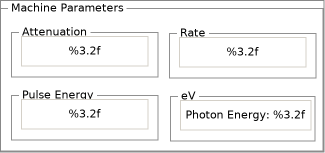
VISUALIZATION BeamParameterStats  // 325x153
VAR_IN_OUT
	BP	:	ST_BeamParams;
END_VAR
    GroupBox (0,0 323x151), "Machine Parameters"
        GroupBox (11,24 147x53), "Attenuation"
            Textfield (10,12 127x30), "%3.2f", text variable: BP.fAtt
        GroupBox (11,87 147x53), "Pulse Energy"
            Textfield (10,12 127x30), "%3.2f", text variable: BP.fPP_mJ
        GroupBox (169,25 147x53), "Rate"
            Textfield (10,12 127x30), "%3.2f", text variable: BP.nRate
        GroupBox (170,88 145x53), "eV"
            Textfield (10,12 131x30), "Photon Energy: %3.2f", text variable: BP.reV
END_VISUALIZATION

(* stored: Version 1.1.0.1, ProductVersion 3.1.4022.12
   Visu BeamParameterStats: Id {2f2224ca-1c7f-0a51-36f0-787385162996} *)
